{attribute 'linkalways'} 
{attribute 'no_explicit_call' := 'This FB is a CLASS and must be accessed using methods or properties'}
{attribute 'enable_dynamic_creation'}
FUNCTION_BLOCK _ETcVnElementType EXTENDS EnumDatatypeBase
VAR
	localData : ETcVnElementType;
	activeData : REFERENCE TO ETcVnElementType;
	enumBaseDatatype : _DINT(localData);
END_VAR

METHOD PRIVATE AddLocalEnumeration
VAR_INPUT
	Enumeration : T_MAXSTRING;
	Value : ETcVnElementType;
END_VAR
AddEnumeration(Enumeration, Value);
END_METHOD

PROPERTY PUBLIC Address : PVOID
GET
Address := ADR(activeData);
END_GET
END_PROPERTY

METHOD PUBLIC ClearReference
VAR_INPUT
END_VAR
activeData REF= localData;
SetBaseDatatypeReference();
END_METHOD

METHOD PUBLIC Clone : I_Datatype
VAR
    pClone : POINTER TO _ETcVnElementType;
END_VAR
pClone := __NEW(_ETcVnElementType(InitialValue := Value));
Clone := pClone^;
END_METHOD

METHOD FB_init : BOOL
VAR_INPUT
	bInitRetains : BOOL; // if TRUE, the retain variables are initialized (warm start / cold start)
	bInCopyCode : BOOL;  // if TRUE, the instance afterwards gets moved into the copy code (online change)
	InitialValue : ETcVnElementType;
END_VAR
localData := InitialValue;
AddBaseDatatype(enumBaseDatatype);
ClearReference();

AddLocalEnumeration('TCVN_ET_SAME_AS_SOURCE', ETcVnElementType.TCVN_ET_SAME_AS_SOURCE);
AddLocalEnumeration('TCVN_ET_USINT', ETcVnElementType.TCVN_ET_USINT);
AddLocalEnumeration('TCVN_ET_SINT', ETcVnElementType.TCVN_ET_SINT);
AddLocalEnumeration('TCVN_ET_UINT', ETcVnElementType.TCVN_ET_UINT);
AddLocalEnumeration('TCVN_ET_INT', ETcVnElementType.TCVN_ET_INT);
AddLocalEnumeration('TCVN_ET_DINT', ETcVnElementType.TCVN_ET_DINT);
AddLocalEnumeration('TCVN_ET_REAL', ETcVnElementType.TCVN_ET_REAL);
AddLocalEnumeration('TCVN_ET_LREAL', ETcVnElementType.TCVN_ET_LREAL);
END_METHOD

PROPERTY PUBLIC Identifier : T_MAXSTRING
GET
Identifier := 'ETcVnElementType';
END_GET
END_PROPERTY

METHOD IsEnumeratorValueEqual : BOOL
VAR_INPUT
	Enumerator : I_KeyValueForwardEnumerator;
END_VAR
VAR
	storedValue : ETcVnElementType;
END_VAR
IF NOT Enumerator.TryGet(storedValue) THEN
	RETURN;
END_IF

IsEnumeratorValueEqual := storedValue = activeData;
END_METHOD

METHOD PUBLIC MakeReferenceTo
VAR_INPUT
	ReferenceTarget : REFERENCE TO ETcVnElementType;
END_VAR
activeData REF= ReferenceTarget;
SetBaseDatatypeReference();
END_METHOD

METHOD PROTECTED SetBaseDatatypeReference
VAR_INPUT
END_VAR
enumBaseDatatype.MakeReferenceTo(activeData);
END_METHOD

PROPERTY PUBLIC Size : UDINT
GET
Size := SIZEOF(activeData);
END_GET
END_PROPERTY

METHOD TryMakeReferenceTo : BOOL
VAR_INPUT
	Target : I_Datatype;
END_VAR
VAR
	targetAsEnum : I_EnumDatatype;
	pTargetData : POINTER TO ETcVnElementType;
END_VAR
IF NOT Target.TryResolveAsEnumDatatype(targetAsEnum) THEN
	RETURN;
END_IF

IF targetAsEnum.Identifier <> Identifier THEN
	RETURN;
END_IF

pTargetData := Target.Address;
activeData REF= pTargetData^;
SetBaseDatatypeReference();
TryMakeReferenceTo := TRUE;
END_METHOD

PROPERTY PUBLIC Value : ETcVnElementType
GET
Value := activeData;
END_GET
SET
activeData := Value;
END_SET
END_PROPERTY

END_FUNCTION_BLOCK

(* stored: Version 1.1.0.1, ProductVersion 3.1.4024.13
   POU _ETcVnElementType: Id {6a2d3efb-f8a4-0528-301c-9864143d5f76}, SpecialFunc None
   Folder Core: Id {3fa38de6-c452-02ac-25d8-caf6d49c5857}
   Folder Protected: Id {74b22dc4-dc85-0f3f-2ce2-7c3a1f91a61f}
   Folder Customize: Id {8df1146c-442c-094e-0bf6-a9c8dc92a2a0}
   Folder Constructor: Id {c6639585-875d-0994-0693-a4a84f47564e}
   Folder Private: Id {f1eb1c9c-a257-0a37-1a46-7ea815335f18}
   Folder Protected: Id {af724463-ad43-0219-339a-8a3813f3e01a}
   Method AddLocalEnumeration: Id {1d251c05-9caa-0d5b-224c-c77e4b15353b}
   Property Address: Id {709393d0-7319-0be9-039e-bc9c6dc1e96a}
   Get Get: Id {cd6b4164-cc06-01d8-1626-0dfb18f3648f}
   Method ClearReference: Id {3a051d4e-8e19-0ebe-2c18-d933d5c94e3f}
   Method Clone: Id {f37be3b4-ed20-0695-04eb-9d37d45f7f97}
   Method FB_init: Id {52d8a469-56a7-08ed-20ec-2cc70e3502d4}
   Property Identifier: Id {36872bcf-355e-0858-3d31-fc343a210a5b}
   Get Get: Id {d08ae839-28da-0ef9-154d-7260360a9631}
   Method IsEnumeratorValueEqual: Id {99654950-0514-00d0-3c6c-1fbf9a68992c}
   Method MakeReferenceTo: Id {ec0613b9-10a2-0fe2-0311-7b4736bd7426}
   Method SetBaseDatatypeReference: Id {7b2da642-347a-020a-2c29-d9930dc3a15d}
   Property Size: Id {65f1e242-8e15-0323-1156-1de3029f106e}
   Get Get: Id {1dded154-4d07-0a98-394b-3f20a276747e}
   Method TryMakeReferenceTo: Id {a5f597e1-f3e0-0e5d-0ac6-4d3358061615}
   Property Value: Id {e845fa0b-d9ba-063f-0807-07bb57e2f19b}
   Get Get: Id {f23e0c73-7c2c-031b-3b71-535842abcd92}
   Set Set: Id {2eab2407-bccb-0e92-21ed-7591ccdc27e2} *)
